(* PLC project SafeLOGIC-1, BrAutomation SafeDESIGNER  4.3.4.4 *)
(* stored: companyURL http://www.br-automation.com, creationDateTime Fri Jun 25 07:58:05 2021 *)

PROGRAM Main
  VAR  (* added by the conversion: wires and edge detectors of the diagram *)
    _SAFEBOOL_TO_BOOL11_OUT : BOOL;
  END_VAR

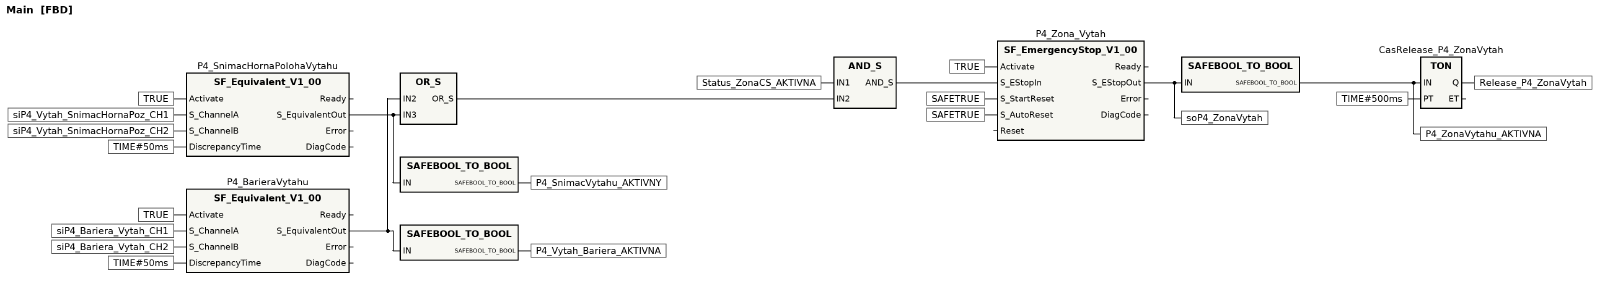
(* FBD diagram, written out as Structured Text *)
P4_BarieraVytahu(Activate := TRUE, S_ChannelA := siP4_Bariera_Vytah_CH1, S_ChannelB := siP4_Bariera_Vytah_CH2, DiscrepancyTime := TIME#50ms);
P4_SnimacHornaPolohaVytahu(Activate := TRUE, S_ChannelA := siP4_Vytah_SnimacHornaPoz_CH1, S_ChannelB := siP4_Vytah_SnimacHornaPoz_CH2, DiscrepancyTime := TIME#50ms);
P4_Zona_Vytah(Activate := TRUE, S_EStopIn := AND_S(Status_ZonaCS_AKTIVNA, OR_S(P4_BarieraVytahu.S_EquivalentOut, P4_SnimacHornaPolohaVytahu.S_EquivalentOut)), S_StartReset := SAFETRUE, S_AutoReset := SAFETRUE);
soP4_ZonaVytah := P4_Zona_Vytah.S_EStopOut;
_SAFEBOOL_TO_BOOL11_OUT := SAFEBOOL_TO_BOOL(P4_Zona_Vytah.S_EStopOut);
P4_ZonaVytahu_AKTIVNA := _SAFEBOOL_TO_BOOL11_OUT;
CasRelease_P4_ZonaVytah(IN := _SAFEBOOL_TO_BOOL11_OUT, PT := TIME#500ms);
Release_P4_ZonaVytah := CasRelease_P4_ZonaVytah.Q;
P4_Vytah_Bariera_AKTIVNA := SAFEBOOL_TO_BOOL(P4_BarieraVytahu.S_EquivalentOut);
P4_SnimacVytahu_AKTIVNY := SAFEBOOL_TO_BOOL(P4_SnimacHornaPolohaVytahu.S_EquivalentOut);
END_PROGRAM
